(* IEC 61131-3 sources: AXOpen/src/components.siem.identification/ctrl/src/IOLink (part 2) *)

(* ---- AxoIOLink_RF200_SwitchAntenna.st ---- *)
USING AXOpen.Components.Abstractions.Drives;
USING AXOpen.Timers;
USING Siemens.Simatic.S71500.DistributedIO;
USING System.Timer;
USING System.Strings;
USING System.Serialization;

NAMESPACE AXOpen.Components.Siem.Identification
    {S7.extern=ReadWrite}
    CLASS PUBLIC AxoIOLink_RF200_SwitchAntenna
        VAR PRIVATE
            statExecuteReq      :	BOOL    :=  FALSE;                          //  State of execute input of last cycle
            statAntStatus       :	BYTE    :=  BYTE#16#0;                      //  Status Byte of antenna
            statState           :	UINT    :=  UINT#0;                         //  Main State Machine Index
            statAnt             :	ARRAY[0..UPPER_BOUND_IO_FIELD] OF BYTE;     //  Received buffer of Antenna data
            statSent            :	ARRAY[0..UPPER_BOUND_IO_FIELD] OF BYTE;     //  Sent buffer for Antenna
            statPresence        :	BOOL    :=  FALSE;                          //  Presence bit. Transponder on field
            statBusy            :	BOOL    :=  FALSE;                          //  TRUE: Job active
            statIoPartError     :	BOOL    :=  FALSE;                          //  TRUE: data in process image is invalid
            statIoPartStatus    :	DWORD   :=  DWORD#16#0;                     //	Status for IO access
            statIOsize          :	INT     :=  INT#0;                          //  Size of the IO-Link Master PII
        END_VAR

        VAR CONSTANT
            IOL_V10                         :	USINT   :=  USINT#10;       //  Identifier IO-Link version 1.0
            IOL_V11                         :	USINT   :=  USINT#11;       //  Identifier IO-Link version 1.1
            LEN_DATA_V10                    :	USINT   :=  USINT#8;        //  Length of user data for IO-Link version 1.0
            LEN_DATA_V11                    :	USINT   :=  USINT#32;       //  Length of user data for IO-Link version 1.1
            UPPER_BOUND_IO_FIELD            :	USINT   :=  USINT#31;       //  Upper bound of Input and Output fields
            STATE_IDLE                      :	UINT    :=  UINT#0;         //  State Machine - Idle State
            STATE_ANTENNA_ON                :	UINT    :=  UINT#1;         //  State Machine - Switch Antenna on
            STATE_ANTENNA_OFF               :	UINT    :=  UINT#2;         //  State Machine - Switch Antenna off
            STATE_READY                     :	UINT    :=  UINT#3;         //  State Machine - Job done
            STATUS_ERROR_IDENT_BLOCK        :	WORD    :=  WORD#16#0001;   //  Error Identification for block internal faults
            STATUS_ERROR_IDENT_RFID         :	WORD    :=  WORD#16#0011;   //  Error Identification for RFID reader faults
            STATUS_NO_JOB                   :	WORD    :=  WORD#16#0000;   //  No job requested
            STATUS_ERROR_TAG_HAS_LEFT       :	WORD    :=  WORD#16#8101;   //  Error - the RFID tag has left the reader
            STATUS_ERROR_STILL_ACTIVE       :	WORD    :=  WORD#16#8102;   //  Error - block still busy, no further request possible
            STATUS_ERROR_LENGTH             :	WORD    :=  WORD#16#8104;   //  Error - requested length is less than 0
            CMD_ANTENNA_ON                  :	BYTE    :=  BYTE#16#00;     //  Command to switsch antenna on
            CMD_ANTENNA_OFF                 :	BYTE    :=  BYTE#16#10;     //  Command to switsch antenna off
            INDEX_ANT_STATUS                :	USINT   :=  USINT#0;        //  Index in Antenna DataField - Status
            INDEX_RFID_ERROR                :	USINT   :=  USINT#1;        //  Index in Antenna DataField - Error
            INDEX_SEND_CMD                  :	USINT   :=  USINT#0;        //  Index in Send DataField - Command

        END_VAR

        METHOD PUBLIC Run
            VAR_INPUT
                execute     :	BOOL    :=  FALSE;          //  Execute function
                antennaState:	BOOL    :=  FALSE;          //  TRUE: activate antenna, FALSE: deactivate antenna
                hwID        :	UINT    :=  UINT#16#0;      //  Hardware identifier of IO-Link communication module
                portAddr    :	INT     :=  INT#0;          //  Start address of port
                version     :	USINT   :=  IOL_V11;        //	IO-Link version of the reader; 11: IO-Link V1.1, 10: IO-Link V1.0
            END_VAR

            VAR_OUTPUT
                done        :	BOOL;       //  TRUE: job done
                busy        :	BOOL;       //  TRUE: Job active
                error       :	BOOL;       //  TRUE: Error has occured
                status      :	DWORD;      //  Error Status
                presence    :	BOOL;       //  TRUE: Transponder on field
            END_VAR

            VAR_TEMP
                tempDone	:   BOOL;   //  Auxiliary tag for done output
                tempError	:   BOOL;   //  Auxiliary tag for error output
                tempStatus  :   DWORD;  //  Auxiliary tag for status output

                tempWord    :   WORD;
                tempData    :   ARRAY[0..255]   OF BYTE;
                tempIndex   :   INT;

            END_VAR

            // INFO HEADER
            //===============================================================================
            // Siemens / (c)Copyright 2022
            //-------------------------------------------------------------------------------
            // Title:            LIOLink_RF200_SwitchAntenna
            // Function:         Switches the antenna of SIMATIC RF200 readers via IO-Link
            // Library:          LIOLink
            // Author:           Siemens Industry Online Support
            // Tested with:      CPU 1513-1 PN FW 2.8
            // Engineering:      TIA Portal V16
            // Restrictions:     --
            // Requirements:     --
            //-------------------------------------------------------------------------------
            // Change log table:
            // Version  | Date       | Expert in charge       | Changes applied
            //----------|------------|------------------------|------------------------------
            // 01.00.00 | 01.07.2013 | Online Support         | First release
            // 01.01.00 | 01.12.2016 | Online Support         | Upgrade to TIA Portal V14
            // 02.00.00 | 01.09.2017 | Online Support         | Upgrade to TIA Portal V14 SP1
            //                                                | Implementation of Programming styleguide
            //                                                | Added support for IO-Link V1.1 readers
            // 02.01.00 | 01.12.2017 | Online Support         | Bug fixes and performance improvements
            // 02.02.00 | 01.03.2020 | Online Support         | Upgrade to TIA Portal V16
            // 02.03.00 | 22.09.2020 | Online Support         | Integrated FB into LIOLink library
            //                                                | Renamed FB to LIOLink_RF200_SwitchAntenna
            //                                                | Combined FBs for IO-Link V1.0 and V1.1
            //                                                | Minor bug fixes
            // 02.04.00 | 04.10.2022 | SUP SPH                | Optimization
            //===============================================================================

            // Check version
            IF version = IOL_V11 THEN                               //determine IO-Link reader version (1.0/1.1) to set offset
                statIOsize := LEN_DATA_V11;
            ELSE
                statIOsize := LEN_DATA_V10;
            END_IF;

            // Get PII

            tempWord := Siemens.Simatic.S71500.DistributedIO.ReadData(TO_WORD(hwID),tempData);
            FOR tempIndex := 0 TO statIOsize - INT#1 DO
                statAnt[tempIndex]   :=  tempData[tempIndex + portAddr];
            END_FOR;

            statAntStatus := statAnt[INDEX_ANT_STATUS];    //status byte
            statPresence := statAntStatus.%X5;    //Presence bit. Transponder on field

            // Check antenna status
            IF statAnt[INDEX_RFID_ERROR] <> BYTE#0 AND statBusy THEN
                tempStatus.%W0 := TO_WORD(statAnt[INDEX_RFID_ERROR]);    //error_BLK
                tempStatus.%W1 := STATUS_ERROR_IDENT_RFID;                    //identifier rfid errors
                statBusy := false;
                tempDone := false;
                tempError := TRUE;
                statState := STATE_IDLE;
            END_IF;

            // Check execute
            // Idle
                IF NOT execute THEN
                    tempDone := false;
                    tempError := false;
                    tempStatus := DWORD#0;
                END_IF;

            // Job executed
                IF execute AND execute <> statExecuteReq THEN //Positive Edge for antenna on
                    statBusy := TRUE;                              //Block active
                    tempDone := FALSE;                             //reset all output parameters
                    tempError := FALSE;
                    tempStatus := STATUS_NO_JOB;
                    IF antennaState THEN                          //if antenna then activate the ANTENNA_ON process
                        statState := STATE_ANTENNA_ON;
                    ELSIF NOT antennaState THEN                   //if not antenna then activate the ANTENNA_OFF process
                        statState := STATE_ANTENNA_OFF;
                    END_IF;

                END_IF;
            statExecuteReq := execute;

        // State machine
            CASE statState OF
                STATE_IDLE:
                    ;

                STATE_ANTENNA_ON:  //Antenna_on
                    //Antenna on process
                    statAntStatus.%X4 := false;                        //Reset Byte 0, bit 4
                    statSent[INDEX_SEND_CMD] := CMD_ANTENNA_ON;

                    FOR tempIndex := INT#0 TO statIOsize - INT#1 DO
                        tempData[tempIndex + portAddr] := statSent[tempIndex];
                    END_FOR;
                    //TODO solve overwriting the outputs in case of several RFID header used with one IOLink master
                    //when SETIO_PART equivalent function is available in AX
                    tempWord := Siemens.Simatic.S71500.DistributedIO.WriteData(TO_WORD(hwID),tempData);

                    IF NOT statIoPartError AND statAnt[INDEX_RFID_ERROR] = BYTE#0 THEN
                        statState := STATE_READY;
                    ELSIF statIoPartError THEN
                        tempError := true;
                        statBusy := FALSE;
                        tempStatus.%W0 :=TO_WORD(statIoPartStatus);//error_BLK
                        tempStatus.%W1 := STATUS_ERROR_IDENT_BLOCK;                    //identifier block errors
                        statState := STATE_IDLE;
                    END_IF;

                STATE_ANTENNA_OFF:
                    //Antenna off process
                    statAntStatus.%X4 := true;                         //set Byte 0, bit 4
                    statSent[INDEX_SEND_CMD] := CMD_ANTENNA_OFF;

                    FOR tempIndex := INT#0 TO statIOsize - INT#1 DO
                        tempData[tempIndex + portAddr] := statSent[tempIndex];
                    END_FOR;
                    //TODO solve overwriting the outputs in case of several RFID header used with one IOLink master
                    //when SETIO_PART equivalent function is available in AX
                    tempWord := Siemens.Simatic.S71500.DistributedIO.WriteData(TO_WORD(hwID),tempData);

                    IF NOT statIoPartError AND statAnt[INDEX_RFID_ERROR] = BYTE#0 THEN
                        IF statAntStatus = CMD_ANTENNA_OFF THEN    //if status_byte=1610 then antenna off
                            statState := STATE_READY;
                        END_IF;
                    ELSIF statIoPartError THEN
                        tempError := true;
                        statBusy := FALSE;
                        tempStatus.%W0 := TO_WORD(statIoPartStatus);    //error_BLK
                        tempStatus.%W1 := STATUS_ERROR_IDENT_BLOCK;   //identifier block errors
                        statState := STATE_IDLE;
                    END_IF;

                STATE_READY:
                    tempDone := true;
                    statBusy := FALSE;
                    statState := STATE_IDLE;
                ELSE
                    statState := STATE_IDLE;
            END_CASE;

            // Update output interface
            done := tempDone;
            busy := statBusy;
            error := tempError;
            status := tempStatus;
            presence := statPresence;
        END_METHOD
    END_CLASS
END_NAMESPACE

(* ---- AxoIOLink_RF200_WriteTag.st ---- *)
USING AXOpen.Components.Abstractions.Drives;
USING AXOpen.Timers;
USING Siemens.Simatic.S71500.DistributedIO;
USING System.Timer;
USING System.Strings;
USING System.Serialization;

NAMESPACE AXOpen.Components.Siem.Identification
    {S7.extern=ReadWrite}
    CLASS PUBLIC AxoIOLink_RF200_WriteTag
        VAR PRIVATE
            instTonR                :	TimeAccumulator;                                //  Tag has left antenna field detection timer
            statState               :	INT     :=  INT#0;                              //	Main State Machine Index
            statTimerIn             :	BOOL    :=  FALSE;                              //  Tag has left antenna field detection timer - Start Tag
            statTimerR              :	BOOL    :=  FALSE;                              //  Tag has left antenna field detection timer - Reset Tag
            statTimerPt             :	TIME    :=  DETECTION_TIME_TAG_OFF_FIELD;       //  Tag has left antenna field detection timer - Detection time
            statStatusByte          :	BYTE    :=  BYTE#16#0;                          //  First received Byte from process image
            statDat                 :	ARRAY[0..UPPER_BOUND_IO_FIELD] OF BYTE;         //  Sent data
            statRecDat              :	ARRAY[0..UPPER_BOUND_IO_FIELD] OF BYTE;         //  Received data
            statPresence            :	BOOL    :=  FALSE;                              //  TRUE: Transponder on field
            statExecuteReq          :	BOOL    :=  FALSE;                              //  State of execute input of last cycle
            statLength              :	DINT    :=  DINT#0;                             //  Length of read Data
            statAddr                :	WORD    :=  WORD#16#0;                          //  Address of Tag
            statWriteOffset         :	INT     :=  INT#0;                              //  Data offset for write function
            statPresenceFf          :	BOOL    :=  FALSE;                              //  Transpnder status of last cycle
            statWriteData           :	ARRAY[0..UPPER_BOUND_MAX_DATA_FIELD] OF BYTE;   //  Data to write to tag
            statDiffToIOsizeNetto   :	INT     :=  INT#0;                              //  Difference to full IO size
            statBytemove            :	INT     :=  INT#0;                              //  Shift value for data
            statDone                :	BOOL    :=  FALSE;                              //  TRUE: job done
            statBusy                :	BOOL    :=  FALSE;                              //  FALSE: no job, TRUE: job in progress
            statError               :	BOOL    :=  FALSE;                              //  FALSE: no error, TRUE: error
            statIoPartError         :	BOOL    :=  FALSE;                              //  TRUE: data in process image is invalid
            statIoPartStatus        :	DWORD   :=  DWORD#16#0;                         //  Status for IO access
            statReturnMoveBlkVar    :	INT     :=  INT#0;                              //  Return Value of Block Move
            statIOsize              :	USINT   :=  USINT#0;                            //  Size of the IO-Link Master PII
            statIOsizeNetto         :	USINT   :=  USINT#0;                            //  Size of the IO-Link Master PAE without header
            statIdentDataLowIndex   :   INT     :=  INT#0;
            statIdentDataHighIndex  :   INT     :=  INT#0;
        END_VAR

        VAR CONSTANT
            IOL_V10                         :	USINT   :=  USINT#10;       //  Identifier IO-Link version 1.0
            IOL_V11                         :	USINT   :=  USINT#11;       //  Identifier IO-Link version 1.1
            LEN_DATA_V10                    :	USINT   :=  USINT#8;        //  Length of user data for IO-Link version 1.0
            LEN_DATA_V11                    :	USINT   :=  USINT#32;       //  Length of user data for IO-Link version 1.1
            UPPER_BOUND_IO_FIELD            :	USINT   :=  USINT#31;       //  Upper bound of Input and Output fields
            UPPER_BOUND_MAX_DATA_FIELD      :	UINT    :=  UINT#1999;      //  Upper bound of the data field of a RFID Tag
            DATA_HEADER_SIZE                :	USINT   :=  USINT#4;    	//  IO-Link Header Size for version 1.0 and 1.1
            STATUS_ERROR_IDENT_BLOCK        :	WORD    :=  WORD#16#0001;   //  Error Identification for block internal faults
            STATUS_ERROR_IDENT_RFID         :	WORD    :=  WORD#16#0011;   //  Error Identification for RFID reader faults
            STATUS_NO_JOB                   :	WORD    :=  WORD#16#0000;   //  No job requested
            STATUS_ERROR_TAG_HAS_LEFT       :	WORD    :=  WORD#16#8101;   //  Error - the RFID tag has left the reader
            STATUS_ERROR_STILL_ACTIVE       :	WORD    :=  WORD#16#8102;   //  Error - block still busy, no further request possible
            STATUS_ERROR_LENGTH             :	WORD    :=  WORD#16#8104;   //  Error - requested length is less than 0
            STATE_IDLE                      :	INT     :=  INT#0;          //  State Machine - Idle State
            STATE_WRITE                     :	INT     :=  INT#2;          //  State Machine - Read Tag
            STATE_TELEGRAM                  :	INT     :=  INT#1;          //  State Machine - Prepare telegram
            STATE_ERROR                     :	INT     :=  INT#3;          //  State Machine - Error State
            DETECTION_TIME_TAG_OFF_FIELD    :	TIME    :=  T#5S;           //  Tag has left antenna field detection time
            CMD_WRITE                       :	BYTE    :=  BYTE#16#01;     //  Command to read data
            CMD_RESET                       :	BYTE    :=  BYTE#16#00;     //  Command to reset
            INDEX_CMD                       :	USINT   :=  USINT#0;        //  Index in DataField - Command
            INDEX_RFID_ERROR                :	USINT   :=  USINT#1;        //  Index in DataField - Error
            INDEX_ADDR_HIGH                 :	USINT   :=  USINT#2;        //  Index in DataField - Address High Byte
            INDEX_ADDR_LOW                  :	USINT   :=  USINT#3;        //  Index in DataField - Address Low Byte
            INDEX_SOURCE_DATA               :	DINT    :=  DINT#4;         //  Index in Data Field - Start of netto Data
            INDEX_REC_STATUS                :	DINT    :=  DINT#0;         //  Index in Received DataField - Status
        END_VAR

        METHOD PUBLIC Run
            VAR_INPUT
                execute     :	BOOL    :=  FALSE;          //  Execute function
                addrTag     :	WORD    :=  WORD#16#0;      //  Start address of data on tag
                length      :	WORD    :=  WORD#16#0;      //  Length of data to be written
                hwID        :	UINT    :=  UINT#16#0;      //  Hardware identifier of IO-Link communication module
                portAddr    :	INT     :=  INT#0;          //  Start address of port
                version     :	USINT   :=  IOL_V11;        //	IO-Link version of the reader; 11: IO-Link V1.1, 10: IO-Link V1.0
                identData   :   REF_TO  ARRAY[*]OF BYTE;    //  Received tag identification data
            END_VAR

            VAR_OUTPUT
                done        :	BOOL;       //  TRUE: job done
                busy        :	BOOL;       //  FALSE: no job, TRUE: job in progress
                error       :	BOOL;       //  FALSE: no error, TRUE: error
                status      :	DWORD;      //  Error Status
                presence    :	BOOL;       //  Tag on antenna field

            END_VAR

            VAR_TEMP
                tempStatus  :   DWORD;  //  Auxiliary tag for status output
                tempWord    :   WORD;
                tempIndex   :   INT;
                tempHWData  :   ARRAY[0..255]   OF BYTE;
            END_VAR

            IF identData = NULL THEN
                // TODO some message
                error := TRUE;
                status  := DWORD#16#FEFE0002;
                RETURN;
            END_IF;

            statIdentDataLowIndex := TO_INT(LOWER_BOUND(identData^, 1));
            statIdentDataHighIndex := TO_INT(UPPER_BOUND(identData^, 1));

            // INFO HEADER
            //===============================================================================
            // Siemens / (c)Copyright 2022
            //-------------------------------------------------------------------------------
            // Title:            LIOLink_RF200_WriteTag
            // Function:         Writes tags on SIMATIC RF200 readers via IO-Link
            // Library:          LIOLink
            // Author:           Siemens Industry Online Support
            // Tested with:      CPU 1513-1 PN FW 2.8
            // Engineering:      TIA Portal V16
            // Restrictions:     --
            // Requirements:     --
            //-------------------------------------------------------------------------------
            // Change log table:
            // Version  | Date       | Expert in charge       | Changes applied
            //----------|------------|------------------------|------------------------------
            // 01.00.00 | 01.03.2015 | Online Support         | First release
            // 01.01.00 | 01.12.2016 | Online Support         | Upgrade to TIA Portal V14
            // 02.00.00 | 01.09.2017 | Online Support         | Upgrade to TIA Portal V14 SP1
            //                                                | Implementation of Programming styleguide
            //                                                | Added support for IO-Link V1.1 readers
            // 02.01.00 | 01.12.2017 | Online Support         | Bug fixes and performance improvements
            // 02.02.00 | 01.03.2020 | Online Support         | Upgrade to TIA Portal V16
            // 02.03.00 | 22.09.2020 | Online Support         | Integrated FB into LIOLink library
            //                                                | Renamed FB to LIOLink_RF200_WriteTag
            //                                                | Combined FBs for IO-Link V1.0 and V1.1
            //                                                | Minor bug fixes
            // 02.04.00 | 04.10.2022 | SUP SPH                | Optimization
            //===============================================================================

            // Check version
            IF version = IOL_V11 THEN   //determine IO-Link reader version (1.0/1.1) to set offsets
                statIOsize := LEN_DATA_V11;
                statIOsizeNetto := LEN_DATA_V11 - DATA_HEADER_SIZE;
            ELSE
                statIOsize := LEN_DATA_V10;
                statIOsizeNetto := LEN_DATA_V10 - DATA_HEADER_SIZE;
            END_IF;

            // Get PII
            // read data from process image
            tempWord := Siemens.Simatic.S71500.DistributedIO.ReadData(TO_WORD(hwID),tempHWData);
            statIoPartStatus := tempWord;
            statIoPartError := tempWord > WORD#0;

            FOR tempIndex := 0 TO statIOsize - INT#1 DO
                statRecDat[tempIndex]   :=  tempHWData[tempIndex + portAddr];
            END_FOR;

            statStatusByte := statRecDat[INDEX_REC_STATUS];    //Status Byte
            statPresence := statStatusByte.%X5;   //Presence bit. Transponder on field

            // Check execute
            // Idle
                IF NOT execute THEN
                    statDone := false;
                    statBusy := false;
                    statError := false;
                    tempStatus := STATUS_NO_JOB;
                END_IF;

            statDiffToIOsizeNetto := TO_INT(length) MOD statIOsizeNetto;
            // Job requested
                IF execute AND execute <> statExecuteReq THEN    //Positive edge for reading of data
                    IF NOT statBusy THEN
                        statAddr := addrTag;    //Transpoder Adress
                        statLength := TO_DINT(length);   //Length of read Data
                        statState := STATE_WRITE;
                        statBusy := TRUE;
                        statDone := FALSE;   //reset all the output parameters
                        statError := FALSE;
                        tempStatus := STATUS_NO_JOB;
                        statWriteOffset := 0;
                        statBytemove := 0;
                        //next step >> send write command
                    ELSE
                        tempStatus.%W0 := STATUS_ERROR_STILL_ACTIVE;    //block is still active
                        tempStatus.%W1 := STATUS_ERROR_IDENT_BLOCK;   //Error identifier for block errors
                        statState := STATE_ERROR;
                    END_IF;
                    IF length < TO_WORD(statIOsizeNetto) THEN
                        tempStatus.%W0 := STATUS_ERROR_LENGTH;    //length too short
                        tempStatus.%W1 := STATUS_ERROR_IDENT_BLOCK;   //identifier rfid errors
                        tempStatus := tempStatus;
                        statState := STATE_ERROR;
                    END_IF;
                END_IF;
            statExecuteReq := execute;

            // Tag presence detection
            IF NOT statPresence AND statPresence <> statPresenceFf THEN    //the tag has left the antenna  field
                IF NOT statDone THEN
                    statTimerIn := true;   //wait 5 sec
                    statTimerR := false;
                END_IF;
            END_IF;
            statPresenceFf := statPresence;
            IF statPresence THEN
                statTimerR := true;
                statTimerIn := false;
            END_IF;

            // State machine
            CASE statState OF
                STATE_IDLE:
                    statWriteOffset := 0;    //offset of puffer must be reseted
                    statBusy := false;
                    statTimerIn := false;

                STATE_WRITE:
                    IF statLength > 0 THEN
                        statDat[INDEX_CMD] := CMD_WRITE;   //Set write command
                        statDat[INDEX_ADDR_HIGH] := statAddr.%B1;    //Adr-H
                        statDat[INDEX_ADDR_LOW] := statAddr.%B0;   //Adr-L

                        FOR tempIndex := INT#0 TO statIdentDataHighIndex - statIdentDataLowIndex - INT#1 DO
                            statWriteData[tempIndex] := identData^[tempIndex + statIdentDataLowIndex];
                        END_FOR;

                        FOR tempIndex := INT#0 TO TO_INT(statIOsizeNetto) - INT#1 DO
                            statDat[INDEX_SOURCE_DATA + tempIndex]  :=  statWriteData[statWriteOffset - statBytemove + tempIndex];
                        END_FOR;
                        //Just statIOsizeNetto Bytes are reserved for every transfer
                    END_IF;
                    IF NOT statIoPartError THEN
                        statState := STATE_TELEGRAM;    //Telegram: Edit the read data
                    END_IF;

                STATE_TELEGRAM:
                    IF statLength > 0 THEN   //Only when length of data>0 can continue
                        IF statStatusByte.%X6 THEN   //IF RFID error has occured
                            tempStatus.%W0 := statRecDat[INDEX_RFID_ERROR];
                            tempStatus.%W1 := STATUS_ERROR_IDENT_RFID;    //Error identifier for RFID errors
                            statState := STATE_ERROR;
                        END_IF;

                        //-------------------------- write command is ready------------------------------------------------//
                        IF statStatusByte.%X7 AND statStatusByte.%X0 THEN
                            IF statRecDat[INDEX_ADDR_HIGH] = statAddr.%B1 AND statRecDat[INDEX_ADDR_LOW] = statAddr.%B0 THEN //received ADR must be ==sent ADR

                                IF NOT statIoPartError THEN
                                    IF statStatusByte.%X7 AND NOT statStatusByte.%X6 THEN
                                        statLength := statLength - statIOsizeNetto;
                                        IF statDiffToIOsizeNetto <> 0 AND statLength < statIOsizeNetto THEN
                                            statBytemove := statIOsizeNetto - statDiffToIOsizeNetto;
                                        END_IF;
                                        //if len is not dividable with statIOsizeNetto the adr offset has to be changed that the last (length < statIOsizeNetto) command is done right
                                        statWriteOffset := statWriteOffset + statIOsizeNetto;                                   //offset must be changed
                                        statAddr := TO_WORD(TO_INT(statAddr) + TO_INT(statIOsizeNetto) - statBytemove);     //Change the ADR on Transponder(statIOsizeNetto Bytes)
                                        statState := STATE_WRITE;                      //Start a new write command
                                    ELSE
                                        statState := STATE_IDLE;
                                    END_IF;
                                ELSE
                                    tempStatus.%W0 := TO_WORD(statIoPartStatus);    //Error has to BLKMOV occured
                                    tempStatus.%W1 := STATUS_ERROR_IDENT_BLOCK;   //functions-Error identifier
                                    statState := STATE_ERROR;
                                END_IF;
                            END_IF;
                        END_IF;

                        FOR tempIndex := INT#0 TO statIOsize - INT#1 DO
                            tempHWData[tempIndex + portAddr] := statDat[tempIndex];
                        END_FOR;
                        //TODO solve overwriting the outputs in case of several RFID header used with one IOLink master
                        //when SETIO_PART equivalent function is available in AX
                        tempWord := Siemens.Simatic.S71500.DistributedIO.WriteData(TO_WORD(hwID),tempHWData);
                        statIoPartStatus := tempWord;
                        statIoPartError := tempWord > WORD#0;

                        IF statIoPartError THEN
                            tempStatus.%W0 := TO_WORD(statIoPartStatus);   //Error has to BLKMOV occured
                            tempStatus.%W1 := STATUS_ERROR_IDENT_BLOCK;   //functions-Error identifier
                            statState := STATE_ERROR;
                        END_IF;

                    ELSE
                        statState := STATE_IDLE;
                        statBusy := false;
                        statDone := TRUE;

                        //Reset write command
                        statDat[INDEX_CMD] := CMD_RESET;

                        FOR tempIndex := INT#0 TO statIOsize - INT#1 DO
                            tempHWData[tempIndex + portAddr] := statDat[tempIndex];
                        END_FOR;
                        //TODO solve overwriting the outputs in case of several RFID header used with one IOLink master
                        //when SETIO_PART equivalent function is available in AX
                        tempWord := Siemens.Simatic.S71500.DistributedIO.WriteData(TO_WORD(hwID),tempHWData);
                        statIoPartStatus := tempWord;
                        statIoPartError := tempWord > WORD#0;
                    END_IF;

                STATE_ERROR:
                    statError := TRUE;
                    statBusy := false;
                    statDone := false;
                    statTimerIn := false;
                    statTimerR := true;
                    statState := STATE_IDLE;

                    //Reset write command
                    statDat[INDEX_CMD] := CMD_RESET;

                    FOR tempIndex := INT#0 TO statIOsize - INT#1 DO
                        tempHWData[tempIndex + portAddr] := statDat[tempIndex];
                    END_FOR;
                    //TODO solve overwriting the outputs in case of several RFID header used with one IOLink master
                    //when SETIO_PART equivalent function is available in AX
                    tempWord := Siemens.Simatic.S71500.DistributedIO.WriteData(TO_WORD(hwID),tempHWData);
                    statIoPartStatus := tempWord;
                    statIoPartError := tempWord > WORD#0;
                ELSE
                    statState := STATE_IDLE;
            END_CASE;

            // Detection timer
            instTonR(signal := statTimerIn,   //this timer will start, if the tag has left the antenna field
                      reset := statTimerR,
                      duration := statTimerPt);
            IF instTonR.output THEN   //error has occured. No tag on field during the 5 sec.
                tempStatus.%W0 := STATUS_ERROR_TAG_HAS_LEFT;  //tag has left the field
                tempStatus.%W1 := STATUS_ERROR_IDENT_BLOCK;   //identifier rfid errors
                statState := STATE_ERROR;
            END_IF;

            // Update output interface
            done := statDone;
            busy := statBusy;
            error := statError;
            status := tempStatus;
            presence := statPresence;

        END_METHOD
    END_CLASS
END_NAMESPACE

(* ---- AxoIOLink_RF200Device.st ---- *)
USING AXOpen.Core;
USING AXOpen.Messaging;
USING AXOpen.Messaging.Static;
USING System.Strings;
USING System.Serialization;
USING Siemens.Simatic.DistributedIO;

NAMESPACE AXOpen.Components.Siem.Identification
    {S7.extern=ReadWrite}
    CLASS PUBLIC AxoIOLink_RF200Device EXTENDS AXOpen.Core.AxoComponent
        VAR PRIVATE
            _infoTimer                  :   AXOpen.Timers.OnDelayTimer;
            _errorTimer                 :   AXOpen.Timers.OnDelayTimer;
            _blink                      :   AXOpen.Timers.AxoBlinker;
            _context                    :   IAxoContext;
            _someTaskIsActive           :   BOOL;

            _HW_ID                      :	UINT    :=  UINT#16#0;
            _portAddr                   :	INT     :=  INT#0;
            _version                    :	USINT   :=  USINT#11;

            _switchAntenna              :   AxoIOLink_RF200_SwitchAntenna;
            _readTag                    :   AxoIOLink_RF200_ReadTag;
            _writeTag                   :   AxoIOLink_RF200_WriteTag;

            _switchAntenna_execute      :   BOOL    :=  FALSE;
            _switchAntenna_antennaState :   BOOL    :=  FALSE;
            _switchAntenna_done         :   BOOL    :=  FALSE;
            _switchAntenna_busy         :   BOOL    :=  FALSE;
            _switchAntenna_error        :   BOOL    :=  FALSE;
            _switchAntenna_status       :   DWORD   :=  DWORD#16#0;
            _switchAntenna_presence     :   BOOL    :=  FALSE;

            _readTag_execute            :   BOOL    :=  FALSE;
            _readTag_addrTag            :	WORD    :=  WORD#16#0;
            _readTag_length             :	WORD    :=  WORD#16#1C;
            _readTag_Data               :   AxoByteArray256;
            _readTag_done               :   BOOL    :=  FALSE;
            _readTag_busy               :   BOOL    :=  FALSE;
            _readTag_error              :   BOOL    :=  FALSE;
            _readTag_status             :   DWORD   :=  DWORD#16#0;
            _readTag_presence           :   BOOL    :=  FALSE;
            _readBuffer                 :   ARRAY[0..255] OF BYTE;

            _writeTag_execute           :   BOOL    :=  FALSE;
            _writeTag_addrTag           :   WORD    :=  WORD#16#0;
            _writeTag_length            :   WORD    :=  WORD#16#1C;
            _writeTag_Data              :   AxoByteArray256;
            _writeTag_done              :   BOOL    :=  FALSE;
            _writeTag_busy              :   BOOL    :=  FALSE;
            _writeTag_error             :   BOOL    :=  FALSE;
            _writeTag_status            :   DWORD   :=  DWORD#16#0;
            _writeTag_presence          :   BOOL    :=  FALSE;
            _writeBuffer                :   ARRAY[0..255] OF BYTE;

            _error                      :   BOOL    :=  FALSE;
            _messageCode                :   ULINT   :=  ULINT#0;
            _lastMessageCode            :   ULINT   :=  ULINT#0;
        END_VAR

        VAR PUBLIC //HEADER

        END_VAR

        VAR PUBLIC //Tasks
            {#ix-attr:[Container(Layout.Wrap)]}
            {#ix-attr:[Group(GroupLayout.GroupBox)]}
            {#ix-attr:[ComponentDetails("Tasks")]}
            {#ix-set:AttributeName = "<#Read tag#>"}
            ReadTagTask : AxoTask;
            {#ix-attr:[ComponentDetails("Tasks")]}
            {#ix-set:AttributeName = "<#Read tag length#>"}
            ReadTag_Length   : WORD;
            {#ix-attr:[ComponentDetails("Tasks")]}
            {#ix-set:AttributeName = "<#Read tag address#>"}
            ReadTag_addrTag         : WORD;

            {#ix-attr:[Group(GroupLayout.GroupBox)]}
            {#ix-attr:[ComponentDetails("Tasks")]}
            {#ix-set:AttributeName = "<#Data read from tag#>"}
            {#ix-attr:[ReadOnly()]}
            {#ix-set:DisplayFormat = "string"}
            ReadTag_Data    : AxoByteArray256;

            {#ix-attr:[Container(Layout.Wrap)]}
            {#ix-attr:[Group(GroupLayout.GroupBox)]}
            {#ix-attr:[ComponentDetails("Tasks")]}
            {#ix-set:AttributeName = "<#Write tag#>"}
            WriteTagTask : AxoTask;
            {#ix-attr:[ComponentDetails("Tasks")]}
            {#ix-set:AttributeName = "<#Write tag lenghth#>"}
            WriteTag_Length   : WORD;
            {#ix-attr:[ComponentDetails("Tasks")]}
            {#ix-set:AttributeName = "<#Write tag address#>"}
            WriteTag_addrTag  : WORD;

            {#ix-attr:[Container(Layout.Wrap)]}
            {#ix-attr:[Group(GroupLayout.GroupBox)]}
            {#ix-attr:[ComponentDetails("Tasks")]}
            {#ix-set:AttributeName = "<#Data to write to tag#>"}
            {#ix-set:DisplayFormat = "string"}
            WriteTag_Data    : AxoByteArray256;

            {#ix-attr:[ComponentDetails("Tasks")]}
            {#ix-set:AttributeName = "<#Restore#>"}
            RestoreTask : AxoTask;
        END_VAR

        VAR PUBLIC //CONFIG
            {#ix-attr:[Container(Layout.Stack)]}
            {#ix-attr:[ComponentDetails("Config")]}
            {#ix-attr:[ReadOnly()]}
            Config  :   Axo_IdentDevice_Config;
        END_VAR

        VAR PUBLIC //STATUS
            {#ix-attr:[Container(Layout.Stack)]}
            {#ix-attr:[ComponentDetails("Status")]}
            {#ix-attr:[ReadOnly()]}
            Status              :   AxoIOLink_RF200Device_Component_Status;
            Messenger           :   AXOpen.Messaging.Static.AxoMessenger;
            TaskMessenger       :   AXOpen.Messaging.Static.AxoMessenger;
            {#ix-attr:[ComponentDetails("Status")]}
            {#ix-attr:[ReadOnly()]}
            {#ix-set:AttributeName = "<#Progress#>"}
            _progress           :   INT := 0;
        END_VAR

        VAR PUBLIC //HardwareDiagnostics
            {#ix-attr:[Container(Layout.Stack)]}
            {#ix-attr:[ComponentDetails("Hardware diagnostics")]}
            {#ix-set:AttributeName = "<#Update diagnostics#>"}
            HardwareDiagnosticsTask :   AXOpen.Io.AxoHardwareDiagnostics;
        END_VAR

        ///<summary>
        /// Runs tasks and logic of this component.
        /// >[!IMPORTANT] This method must or one of its overloads be called cyclically.
        ///</summary>
        METHOD PUBLIC Run
            VAR_INPUT
                inParent    :   IAxoObject;
                HW_ID       :	UINT    :=  UINT#16#0;      //	Logic IO address of the IO-Link Master
                portAddr    :	INT     :=  INT#0;          //  Start address of port
                version     :	USINT   :=  USINT#11;       //	IO-Link version of the reader; 11: IO-Link V1.1, 10: IO-Link V1.0
            END_VAR
            VAR
                i : INT;
            END_VAR

            SUPER.Run(inParent);

            Messenger.Serve(THIS);

            Messenger.ActivateOnCondition(ULINT#700,inParent = NULL, eAxoMessageCategory#ProgrammingError);
            Messenger.ActivateOnCondition(ULINT#701,HW_ID = UINT#0, eAxoMessageCategory#ProgrammingError);

            IF inParent = NULL THEN
                Status.Error.Id := UINT#700;
                RETURN;
            ELSIF HW_ID = UINT#0 THEN
                Status.Error.Id := UINT#701;
                RETURN;
            END_IF;

            _HW_ID      :=  HW_ID;
            _portAddr   :=  portAddr;
            _version    :=  version;

            //*********************************************
            // THIS.Execute();
            //*************Execute inline******************

            _switchAntenna.Run( execute         :=      _switchAntenna_execute,
                                antennaState    :=      _switchAntenna_antennaState,
                                hwID            :=      _HW_ID,
                                portAddr        :=      _portAddr,
                                version         :=      _version,
                                done            =>      _switchAntenna_done,
                                busy            =>      _switchAntenna_busy,
                                error           =>      _switchAntenna_error,
                                status          =>      _switchAntenna_status,
                                presence        =>      _switchAntenna_presence);

            _readTag.Run(   execute     :=  _readTag_execute,
                            addrTag     :=  _readTag_addrTag,
                            length      :=  _readTag_length,
                            hwID        :=  _HW_ID,
                            portAddr    :=  _portAddr,
                            version     :=  _version,
                            identData   :=  REF(_readBuffer),
                            done        =>  _readTag_done,
                            busy        =>  _readTag_busy,
                            error       =>  _readTag_error,
                            status      =>  _readTag_status,
                            presence    =>  _readTag_presence);

            _writeTag.Run(  execute     :=  _writeTag_execute,
                            addrTag     :=  _writeTag_addrTag,
                            length      :=  _writeTag_length,
                            hwID        :=  _HW_ID,
                            portAddr    :=  _portAddr,
                            version     :=  _version,
                            identData   :=  REF(_writeBuffer),
                            done        =>  _writeTag_done,
                            busy        =>  _writeTag_busy,
                            error       =>  _writeTag_error,
                            status      =>  _writeTag_status,
                            presence    =>  _writeTag_presence);

            Status.Antenna_status     :=  _switchAntenna_status;
            Status.ReadTag_status     :=  _readTag_status;
            Status.WriteTag_status    :=  _writeTag_status;

            Messenger.ActivateOnCondition(TO_ULINT(DWORD#16#FEFE0001),_readTag_status = DWORD#16#FEFE0001, eAxoMessageCategory#ProgrammingError);
            Messenger.ActivateOnCondition(TO_ULINT(DWORD#16#FEFE0002),_writeTag_status = DWORD#16#FEFE0002, eAxoMessageCategory#ProgrammingError);

            _error := FALSE;
            IF _switchAntenna_error THEN
                _error := TRUE;
                IF _messageCode = ULINT#0 THEN
                    _messageCode := TO_ULINT(_switchAntenna_status);
                END_IF;
            ELSIF _readTag_error THEN
                _error := TRUE;
                IF _messageCode = ULINT#0 THEN
                    _messageCode := TO_ULINT(_readTag_status);
                END_IF;
            ELSIF _writeTag_error THEN
                _error := TRUE;
                IF _messageCode = ULINT#0 THEN
                    _messageCode := TO_ULINT(_writeTag_status);
                END_IF;
            END_IF;

            Messenger.ActivateOnCondition(_messageCode, _error AND _messageCode = _lastMessageCode ,eAxoMessageCategory#Error);

            // IF NOT Messenger.IsActive THEN
            IF Messenger.MessengerState = eAxoMessengerState#Idle THEN
                IF _error THEN
                    _lastMessageCode := _messageCode;
                    RETURN;
                ELSE
                    _messageCode := ULINT#0;
                END_IF;
            END_IF;

            //*******************************************
            _context := THIS.GetContext();

            //*************INITIALIZATION****************
            // RestoreTask.Run(THIS);
            // ReadTagTask.Run(THIS);
            // WriteTagTask.Run(THIS);
            // HardwareDiagnosticsTask.Run(THIS);

            //*******************************************
            //********************Diagnostics************
            HardwareDiagnosticsTask.Run(THIS,_HW_ID);
            //*******************************************

            //*************RESTORE***********************
            RestoreTask.SetIsDisabled(FALSE);
            IF RestoreTask.Execute(THIS) THEN
                THIS.Restore();
            END_IF;
            //*******************************************

            //*************ReadTask**********************
            ReadTagTask.SetIsDisabled(FALSE);
            IF ReadTagTask.StartTriggered() THEN
                Status.Action.Id :=  UINT#100;
            END_IF;
            Messenger.ActivateOnCondition(ULINT#100,ReadTagTask.IsBusy(), eAxoMessageCategory#Info);
            Messenger.ActivateOnCondition(ULINT#101,ReadTagTask.IsDone(), eAxoMessageCategory#Info);
            IF ReadTagTask.Execute(THIS) THEN
                _blink.Blink(Context := _context, inOnTime:=T#500MS,inOffTime:=T#500MS);
                IF _progress = 0 THEN
                    Status.Error.Id :=  UINT#0;
                    TaskMessenger.Restore();
                    THIS.CallTimers(FALSE);
                    _switchAntenna_execute := FALSE;
                    _readTag_execute := FALSE;
                    _writeTag_execute := FALSE;
                    FOR i := INT#0 TO INT#255 DO
                        _readTag_Data.Data[i] := BYTE#0;
                    END_FOR;
                    _readTag_Data.ToggleDataChangedFlag();
                    _progress := 300;
                END_IF;

                IF _progress = 300 THEN
                    IF _infoTimer.output THEN
                        TaskMessenger.Activate( UINT#500, eAxoMessageCategory#Warning);
                        Status.Error.Id :=      UINT#500;
                    END_IF;

                    _switchAntenna_execute      :=  TRUE;
                    _switchAntenna_antennaState :=  TRUE;

                    IF _switchAntenna_done THEN
                        THIS.CallTimers(FALSE);
                        _progress:=301;
                    END_IF;
                    ReadTagTask.ThrowWhen(_switchAntenna_error,'Error when switching the antena On' );
                END_IF;

                IF _progress = 301 THEN
                    IF _infoTimer.output THEN
                        TaskMessenger.Activate( UINT#501, eAxoMessageCategory#Warning);
                        Status.Error.Id :=      UINT#501;
                    END_IF;

                    _switchAntenna_execute      :=  FALSE;

                    IF( NOT _switchAntenna_done) THEN
                        THIS.CallTimers(FALSE);
                        _progress:=302;
                     END_IF;
                END_IF;

                IF _progress = 302 THEN
                    IF _infoTimer.output THEN
                        TaskMessenger.Activate( UINT#502, eAxoMessageCategory#Warning);
                        Status.Error.Id :=      UINT#502;
                    END_IF;

                    IF(_switchAntenna_presence) THEN
                        THIS.CallTimers(FALSE);
                        _progress:=303;
                     END_IF;
                END_IF;

                IF _progress = 303 THEN
                    IF _infoTimer.output THEN
                        TaskMessenger.Activate( UINT#503, eAxoMessageCategory#Warning);
                        Status.Error.Id :=      UINT#503;
                    END_IF;

                    _readTag_execute := TRUE;

                    IF(_readTag_done) THEN
                        THIS.CallTimers(FALSE);
                        _progress:=304;
                     END_IF;
                     ReadTagTask.ThrowWhen(_readTag_error,'Error reading tag');
                    END_IF;

                IF _progress = 304 THEN
                    IF _infoTimer.output THEN
                        TaskMessenger.Activate( UINT#504, eAxoMessageCategory#Warning);
                        Status.Error.Id :=      UINT#504;
                    END_IF;

                    FOR i := 0 TO TO_INT(_readTag_length) - INT#1 DO
                        _readTag_Data.Data[i] := _readBuffer[i];
                    END_FOR;

                    _readTag_execute           :=  FALSE;

                    IF NOT _readTag_done THEN
                        THIS.CallTimers(FALSE);
                        _progress:=305;
                    END_IF;
                END_IF;

                IF _progress = 305 THEN
                    _readTag_Data.ToggleDataChangedFlag();
                    ReadTagTask.DoneWhen(TRUE);
                    THIS.CallTimers(FALSE);
                    _progress := 0;
                END_IF;

                THIS.CallTimers(TRUE);
                ReadTagTask.ThrowWhen(_errorTimer.output );
                Status.Action.Id := TO_UINT(_progress);
            END_IF;
            IF ReadTagTask.DoneReached() THEN
                Status.Action.Id :=  UINT#101;
                Status.Error.Id :=  UINT#0;
            ELSIF ReadTagTask.ErrorOccured() THEN
                Status.Action.Id :=  UINT#10000;
                Status.Error.Id  :=  UINT#10000;
            ELSIF ReadTagTask.AbortTriggered()THEN
                Status.Action.Id :=  UINT#10001;
                Status.Error.Id  :=  UINT#10001;
            END_IF;
            Messenger.ActivateOnCondition(ULINT#10000,ReadTagTask.HasError(), eAxoMessageCategory#Error);
            Messenger.ActivateOnCondition(ULINT#10001,ReadTagTask.IsAborted(), eAxoMessageCategory#Error);
            Messenger.ActivateOnCondition(ULINT#102,ReadTagTask.RestoreTriggered() , eAxoMessageCategory#Error);
            IF ReadTagTask.RestoreTriggered() AND _progress >= 300 AND _progress <= 309  THEN
                Status.Action.Id :=  UINT#102;
                _progress := 0;
            END_IF;
            //*******************************************

            //***********WriteTask***********************
            WriteTagTask.SetIsDisabled(FALSE);
            IF WriteTagTask.StartTriggered() THEN
                Status.Action.Id :=  UINT#120;
            END_IF;
            Messenger.ActivateOnCondition(ULINT#120,WriteTagTask.IsBusy(), eAxoMessageCategory#Info);
            Messenger.ActivateOnCondition(ULINT#121,WriteTagTask.IsDone(), eAxoMessageCategory#Info);
            IF WriteTagTask.Execute(THIS) THEN
                _blink.Blink(Context := _context, inOnTime:=T#500MS,inOffTime:=T#500MS);
                IF _progress = 0 THEN
                    Status.Error.Id :=  UINT#0;
                    TaskMessenger.Restore();
                    THIS.CallTimers(FALSE);
                    _switchAntenna_execute := FALSE;
                    _readTag_execute := FALSE;
                    _writeTag_execute := FALSE;
                    _progress := 320;
                END_IF;

                IF _progress = 320 THEN
                    IF _infoTimer.output THEN
                        TaskMessenger.Activate( UINT#520, eAxoMessageCategory#Warning);
                        Status.Error.Id :=      UINT#520;
                    END_IF;

                    FOR i := INT#0 TO TO_INT(_writeTag_length) - INT#1 DO
                        _writeBuffer[i] := _writeTag_Data.Data[i];
                    END_FOR;

                    _switchAntenna_execute      :=  TRUE;
                    _switchAntenna_antennaState :=  TRUE;

                    IF _switchAntenna_done THEN
                        THIS.CallTimers(FALSE);
                        _progress:=321;
                    END_IF;
                    WriteTagTask.ThrowWhen(_switchAntenna_error,'Error when switching the antena On' );
                END_IF;

                IF _progress = 321 THEN
                    IF _infoTimer.output THEN
                        TaskMessenger.Activate( UINT#521, eAxoMessageCategory#Warning);
                        Status.Error.Id :=      UINT#521;
                    END_IF;

                    _switchAntenna_execute      :=  FALSE;

                    IF( NOT _switchAntenna_done) THEN
                        THIS.CallTimers(FALSE);
                        _progress:=322;
                     END_IF;
                END_IF;

                IF _progress = 322 THEN
                    IF _infoTimer.output THEN
                        TaskMessenger.Activate( UINT#522, eAxoMessageCategory#Warning);
                        Status.Error.Id :=      UINT#522;
                    END_IF;

                    IF(_switchAntenna_presence) THEN
                        THIS.CallTimers(FALSE);
                        _progress:=323;
                     END_IF;
                END_IF;

                IF _progress = 323 THEN
                    IF _infoTimer.output THEN
                        TaskMessenger.Activate( UINT#523, eAxoMessageCategory#Warning);
                        Status.Error.Id :=      UINT#523;
                    END_IF;

                    _writeTag_execute := TRUE;

                    IF(_writeTag_done) THEN
                        THIS.CallTimers(FALSE);
                        _progress:=324;
                     END_IF;
                     WriteTagTask.ThrowWhen(_writeTag_error,'Error writing tag');
                    END_IF;

                IF _progress = 324 THEN
                    IF _infoTimer.output THEN
                        TaskMessenger.Activate( UINT#524, eAxoMessageCategory#Warning);
                        Status.Error.Id :=      UINT#524;
                    END_IF;

                    _writeTag_execute           :=  FALSE;

                    IF NOT _writeTag_done THEN
                        THIS.CallTimers(FALSE);
                        _progress:=325;
                    END_IF;
                END_IF;

                IF _progress = 325 THEN
                    WriteTagTask.DoneWhen(TRUE);
                    THIS.CallTimers(FALSE);
                    _progress := 0;
                END_IF;

                THIS.CallTimers(TRUE);
                WriteTagTask.ThrowWhen(_errorTimer.output);
                Status.Action.Id := TO_UINT(_progress);
            END_IF;
            IF WriteTagTask.DoneReached() THEN
                Status.Action.Id :=  UINT#121;
                Status.Error.Id :=  UINT#0;
            ELSIF WriteTagTask.ErrorOccured() THEN
                Status.Action.Id :=  UINT#10020;
                Status.Error.Id  :=  UINT#10020;
            ELSIF WriteTagTask.AbortTriggered() THEN
                Status.Action.Id :=  UINT#10021;
                Status.Error.Id  :=  UINT#10021;
            END_IF;
            Messenger.ActivateOnCondition(ULINT#10020,WriteTagTask.HasError(), eAxoMessageCategory#Error);
            Messenger.ActivateOnCondition(ULINT#10021,WriteTagTask.IsAborted(), eAxoMessageCategory#Error);
            Messenger.ActivateOnCondition(ULINT#122,WriteTagTask.RestoreTriggered() , eAxoMessageCategory#Error);
            IF WriteTagTask.RestoreTriggered() AND _progress >= 320 AND _progress <= 339  THEN
                Status.Action.Id :=  UINT#122;
                _progress := 0;
            END_IF;
            //*******************************************

            //*******************************************
        END_METHOD

        METHOD PROTECTED OVERRIDE ManualControl
            _readTag_addrTag    :=  ReadTag_addrTag;
            _readTag_Length     :=  ReadTag_Length;
            ReadTag_Data        :=  _readTag_Data;
            _writeTag_Data      :=  WriteTag_Data;
            _writeTag_addrTag   :=  WriteTag_addrTag;
            _writeTag_Length    :=  WriteTag_Length;
        END_METHOD

        ///<summary>
        /// Restores this component into intial state.
        ///</summary>
        METHOD PUBLIC OVERRIDE Restore
            ReadTagTask.Restore();
            WriteTagTask.Restore();
            Status.Action.Id :=  UINT#50;
            RestoreTask.DoneWhen(TRUE);
        END_METHOD

        ///<summary>
        /// Reads the data from the transponder into the array of byte.
        ///</summary>
        METHOD PUBLIC ReadTag : IAxoTaskState
            VAR_INPUT
                Address     :   WORD;
                Length      :   WORD;
                Data        :   REF_TO AxoByteArray256;
            END_VAR
            VAR
                _i              :   INT;
            END_VAR

            IF Data = NULL THEN
                RETURN;
            END_IF;

            _readTag_addrTag    :=  Address;
            _readTag_Length     :=  Length;

            IF ReadTagTask.IsFirstExecutionCycle() THEN
                FOR _i := INT#0 TO INT#255 DO
                    Data^.Data[_i] := BYTE#0;
                END_FOR;
            END_IF;

            ReadTag := ReadTagTask.Invoke(THIS);

            IF ReadTagTask.DoneReached() THEN
                FOR _i := INT#0 TO TO_INT(Length) - INT#1 DO
                    Data^.Data[_i] := _readTag_Data.Data[_i];
                END_FOR;
            END_IF;
        END_METHOD

        ///<summary>
        /// Reads the data from the transponder into the string.
        ///</summary>
        METHOD PUBLIC ReadTag : IAxoTaskState
            VAR_INPUT
                Address     :   WORD;
                Length      :   WORD;
            END_VAR
            VAR_OUTPUT
                Data            :   STRING;
            END_VAR
            VAR
                _i              :   INT;
                _data           :   ARRAY[0..255] OF BYTE;
            END_VAR

            _readTag_addrTag    :=  Address;
            _readTag_Length     :=  Length;

            IF ReadTagTask.IsFirstExecutionCycle() THEN
                Data := '';
             END_IF;

            ReadTag := ReadTagTask.Invoke(THIS);

            IF ReadTagTask.DoneReached() THEN
                _data[0]    :=  TO_BYTE(Length);
                FOR _i := INT#1 TO TO_INT(Length)  DO
                    _data[_i] := _readTag_Data.Data[_i - INT#1];
                END_FOR;
                Deserialize(UINT#0,_data,Data);
            END_IF;
        END_METHOD

        ///<summary>
        /// Writes the data from the array of byte into the transponder.
        ///</summary>
        METHOD PUBLIC WriteTag : IAxoTaskState
            VAR_INPUT
                Data        :   REF_TO AxoByteArray256;
                Address     :   WORD;
                Lenght      :   WORD;
            END_VAR

            IF Data = NULL THEN
                RETURN;
            END_IF;

            _writeTag_Data      :=  Data^;
            _writeTag_addrTag   :=  Address;
            _writeTag_Length    :=  Lenght;

            WriteTag := WriteTagTask.Invoke(THIS);
        END_METHOD

        ///<summary>
        /// Writes the data from the string into the transponder.
        ///</summary>
        METHOD PUBLIC WriteTag : IAxoTaskState
            VAR_INPUT
                Data            :   STRING;
                Address         :   WORD;
            END_VAR
            VAR
                _i              :   INT;
                _data           :   ARRAY[0..256] OF BYTE;
            END_VAR
            Serialize(UINT#0,Data,_data);
            FOR _i := INT#0 TO LengthOf(Data) DO
                _writeTag_Data.Data[_i] := _data[_i + INT#1];
            END_FOR;

            _writeTag_addrTag   :=  Address;
            _writeTag_length  :=  TO_WORD(LengthOf(Data));

            WriteTag := WriteTagTask.Invoke(THIS);
        END_METHOD

        METHOD PRIVATE CallTimers
            VAR_INPUT
                signal : BOOL;
            END_VAR

            _infoTimer.OnDelay(THIS, signal AND Config.InfoTime > LT#0S ,Config.InfoTime);
            _errorTimer.OnDelay(THIS, signal AND Config.ErrorTime > LT#0S , Config.ErrorTime);

        END_METHOD
    END_CLASS
END_NAMESPACE
